(* PLC project Untitled1, Beckhoff Automation GmbH TwinCAT PLC Control 3.5.13.21 *)
(* stored: creationDateTime 2026-03-04T12:40:17.5987306, modificationDateTime 2026-03-04T12:40:17.5997101 *)

(* global variable list GVL_PLC *)
{attribute 'qualified_only'}
VAR_GLOBAL
	(*0x0001 = Link error
	0x0002 = I/O locked after link error (I/O reset required)
	0x0004 = Link error (redundancy adapter)
	0x0008 = Missing one frame (redundancy mode)
	0x0010 = Out of send resources (I/O reset required)
	0x0020 = Watchdog triggered
	0x0040 = Ethernet driver (miniport) not found
	0x0080 = I/O reset active
	0x0100 = At least one device in 'INIT' state
	0x0200 = At least one device in 'PRE-OP' state
	0x0400 = At least one device in 'SAFE-OP' state
	0x0800 = At least one device indicates an error state
	0x1000 = DC not in sync*)
	{attribute 'OPC.UA.DA' := '1'}
	SystemStatus : UINT;
	
	{attribute 'OPC.UA.DA' := '1'}
	AllPartitiantsPresent : BOOL;
		
	//CANCloseState. True if ok
	{attribute 'OPC.UA.DA' := '1'}
	CANCloseState : BOOL;
	
	//Compiler timestamp
	{attribute 'OPC.UA.DA' := '1'}
	AppTimestamp : DT;

	//Current plc version
	{attribute 'OPC.UA.DA' := '1'}
	AppVersion : STRING;
	
	//Current plc version is released
	{attribute 'OPC.UA.DA' := '1'}
	IsReleased :BOOL;

	{attribute 'OPC.UA.DA' := '1'}
	SomeOtherNode : BOOL;
END_VAR
VAR_GLOBAL CONSTANT
	iExpectedNumberOfPartitiants : UINT := 35; //set Number of Expected Ethercat Partitians
END_VAR
